TYPE CollectionSize : DINT(1..2147483647); END_TYPE

(* stored: Version 1.1.0.1
   DUT CollectionSize: Id {93965e5a-bfbc-439f-a2f4-ec0b6924c93a} *)
